PROGRAM PRG_XX_Visualization_Variables
VAR
	

END_VAR

bRemote := IN_bRemote ;
bAutoCrossCutSingle := NOT IN_bAutoCrossCutDouble ;
bAutoCrossCutDouble := IN_bAutoCrossCutDouble ;
bZAxisSlow := IN_bZaxisSlow ;
bZAxisMed := NOT IN_bZaxisSlow AND NOT IN_bZaxisFast ;
bZAxisFast := IN_bZaxisFast ;
bTrtCCW := OUT_bTrtContactor AND OUT_bTrtCrgLH ;
bTrtCW := OUT_bTrtContactor AND OUT_bTrtCrgRH ;
bCrgLH := OUT_bCrgContactor AND OUT_bTrtCrgLH ;
bCrgRH := OUT_bCrgContactor AND OUT_bTrtCrgRH ;
bTeachLeft := IN_bTeachLeft ;
bTeachRight := IN_bTeachRight ;

END_PROGRAM

(* stored: Version 1.1.0.1, ProductVersion 3.1.4024.12
   POU PRG_XX_Visualization_Variables: Id {656fc471-b434-4e21-9c55-dbe503452562}, SpecialFunc None *)
